INTERFACE I_MotionInterlocksLimSw EXTENDS I_MotionInterlocksGeneric, I_LimSwStatus

END_INTERFACE

(* stored: Version 1.1.0.1
   Itf I_MotionInterlocksLimSw: Id {fcbaac2d-99c6-4ac2-b5e1-5ff84c410a2f} *)
